(* CoDeSys 2.3 export: FILLSPACESTRING.EXP *)

(* POU FUNv1/FillSpaceString, ST *)
(*заполняет строку пробелами до указанной длины*)
FUNCTION FillSpaceString : STRING
VAR_INPUT
    str:   STRING;
    index: UINT;
END_VAR
VAR
    i:     INT;
    ii:    INT;
END_VAR
ii := LEN(str);
FillSpaceString := str;
FOR i := ii TO index - 1 DO
    FillSpaceString := CONCAT(FillSpaceString, ' ');
END_FOR
END_FUNCTION
